Universal Robots PolyScope program: reciprocal_p2_1.urp

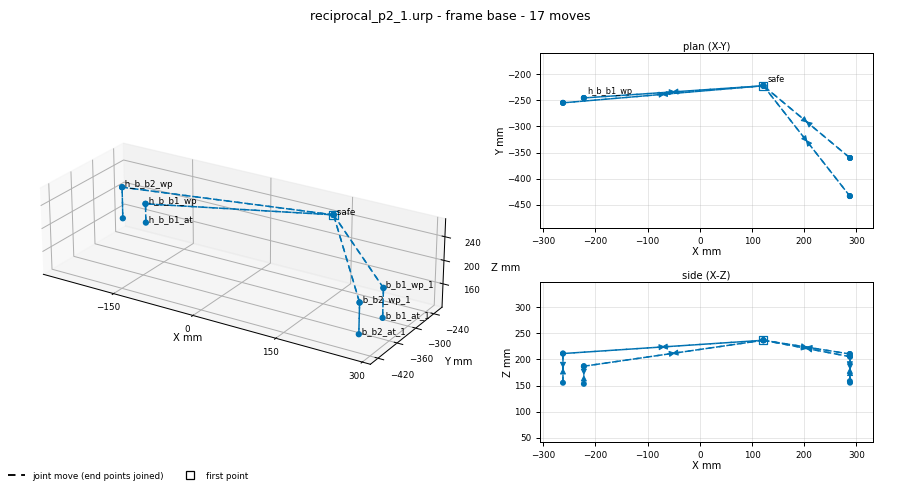
[picture p0: tool path of reciprocal_p2_1.urp in frame base, 17 of 17 moves have a stored position in this frame; points joined in program order, loops and branches not executed]
Program reciprocal_p2_1 (installation=default directory=/programs/ITER createdIn=5.3.1.64192 lastSavedIn=5.3.1.64192 robotSerialNumber=20195300365)
Calibrated DH parameters: a=[-0.000093, -0.190649, -0.212673, 0.000091, -0.000205, 0]; d=[0.151591, 44.061648, -42.488068, -1.442789, 0.085322, 0.091911]; alpha=[1.570082, -0.003447, 0.007513, 1.572293, -1.571904, 0]; deltaTheta=[0, -0.672656, 0.728185, -0.055522, 0.000005, 0]
Robot Program (runOnlyOnce=true)
  URCap Gripper Activate (Robotiq_Grippers, Robotiq Inc.) dataModel(ResetAndActivateKey=false)
  URCap Gripper (Robotiq_Grippers, Robotiq Inc.) dataModel(position=50.0, force=100.0, speed=100.0, positionInDouble=50.0, forceInDouble=100.0, speedInDouble=100.0, slaveIds=[9], blocking=true)
  Folder Base
    MoveJ speed 60 deg/s, acceleration 80 deg/s^2 (useActiveTCP=true) feature=Base
      Waypoint safe: motionParameters(blendRadius=0.075); TCP in base x=121.882 y=-222.057 z=236.793 mm, rx=2.2146 ry=2.209 rz=-0.0386 rad; joints [-29.832, -71.908, -123.399, -74.268, 88.825, -209.331] deg
      Waypoint b_b1_wp_1: TCP in base x=287.856 y=-360.368 z=205.358 mm, rx=2.2407 ry=2.1786 rz=-0.0803 rad; joints [-34.358, -127.348, -66.069, -76.253, 87.212, -212.545] deg
      Waypoint b_b1_at_1: TCP in base x=287.864 y=-360.357 z=155.443 mm, rx=2.2407 ry=2.1786 rz=-0.0802 rad; joints [-34.375, -131.385, -73.13, -65.157, 87.19, -212.499] deg
      URCap Gripper (Robotiq_Grippers, Robotiq Inc.) dataModel(position=100.0, force=100.0, speed=100.0, positionInDouble=100.0, forceInDouble=100.0, speedInDouble=100.0, slaveIds=[9], blocking=true)
      Waypoint b_b1_wp_2: TCP in base x=287.856 y=-360.368 z=205.358 mm, rx=2.2407 ry=2.1786 rz=-0.0803 rad; joints [-34.358, -127.348, -66.069, -76.253, 87.212, -212.545] deg
      Waypoint safe: motionParameters(blendRadius=0.075); TCP in base x=121.882 y=-222.057 z=236.793 mm, rx=2.2146 ry=2.209 rz=-0.0386 rad; joints [-29.832, -71.908, -123.399, -74.268, 88.825, -209.331] deg
      Waypoint h_b_b1_wp: TCP in base x=-222.187 y=-245.349 z=187.06 mm, rx=-3.1315 ry=0.0204 rz=0.0123 rad; joints [-108.957, -99.116, -113.081, -58.146, 89.665, -197.782] deg
      Waypoint h_b_b1_at: TCP in base x=-222.188 y=-245.348 z=153.24 mm, rx=-3.1314 ry=0.0204 rz=0.0122 rad; joints [-108.969, -104.391, -117.643, -48.312, 89.612, -197.745] deg
      URCap Gripper (Robotiq_Grippers, Robotiq Inc.) dataModel(position=50.0, force=100.0, speed=100.0, positionInDouble=50.0, forceInDouble=100.0, speedInDouble=100.0, slaveIds=[9], blocking=true)
      Waypoint h_b_b1_wp: TCP in base x=-222.187 y=-245.349 z=187.06 mm, rx=-3.1315 ry=0.0204 rz=0.0123 rad; joints [-108.957, -99.116, -113.081, -58.146, 89.665, -197.782] deg
    MoveJ speed 60 deg/s, acceleration 80 deg/s^2 (useActiveTCP=true) feature=Base
      Waypoint safe: motionParameters(blendRadius=0.075); TCP in base x=121.882 y=-222.057 z=236.793 mm, rx=2.2146 ry=2.209 rz=-0.0386 rad; joints [-29.832, -71.908, -123.399, -74.268, 88.825, -209.331] deg
      Waypoint b_b2_wp_1: TCP in base x=287.521 y=-433.433 z=210.514 mm, rx=2.2195 ry=2.211 rz=-0.063 rad; joints [-41.44, -147.038, -28.419, -94.163, 87.942, -221.217] deg
      Waypoint b_b2_at_1: TCP in base x=287.518 y=-433.44 z=158.432 mm, rx=2.2196 ry=2.211 rz=-0.063 rad; joints [-41.471, -147.777, -41.016, -80.833, 87.944, -221.148] deg
      URCap Gripper (Robotiq_Grippers, Robotiq Inc.) dataModel(position=100.0, force=100.0, speed=100.0, positionInDouble=100.0, forceInDouble=100.0, speedInDouble=100.0, slaveIds=[9], blocking=true)
      Waypoint b_b2_wp_2: TCP in base x=287.521 y=-433.433 z=210.514 mm, rx=2.2195 ry=2.211 rz=-0.063 rad; joints [-41.44, -147.038, -28.419, -94.163, 87.942, -221.217] deg
      Waypoint safe: motionParameters(blendRadius=0.075); TCP in base x=121.882 y=-222.057 z=236.793 mm, rx=2.2146 ry=2.209 rz=-0.0386 rad; joints [-29.832, -71.908, -123.399, -74.268, 88.825, -209.331] deg
      Waypoint h_b_b2_wp: TCP in base x=-262.196 y=-254.726 z=211.351 mm, rx=-3.0605 ry=0.0443 rz=-0.0223 rad; joints [-114.749, -105.359, -96.042, -73.109, 89.199, -202.734] deg
      Waypoint h_b_b2_at: TCP in base x=-262.208 y=-254.718 z=155.33 mm, rx=-3.0605 ry=0.0443 rz=-0.0223 rad; joints [-114.774, -111.736, -104.192, -58.581, 89.146, -202.674] deg
      URCap Gripper (Robotiq_Grippers, Robotiq Inc.) dataModel(position=50.0, force=100.0, speed=100.0, positionInDouble=50.0, forceInDouble=100.0, speedInDouble=100.0, slaveIds=[9], blocking=true)
      Waypoint h_b_b2_wp: TCP in base x=-262.196 y=-254.726 z=211.351 mm, rx=-3.0605 ry=0.0443 rz=-0.0223 rad; joints [-114.749, -105.359, -96.042, -73.109, 89.199, -202.734] deg
  MoveJ speed 60 deg/s, acceleration 80 deg/s^2 (useActiveTCP=true) feature=Base
    Waypoint safe_end: TCP in base x=121.882 y=-222.057 z=236.793 mm, rx=2.2146 ry=2.209 rz=-0.0386 rad; joints [-29.832, -71.908, -123.399, -74.268, 88.825, -209.331] deg
